// TwinCAT 3 PLC project Untitled1
// ProgramVersion: 3.1.4024.12
// libraries:
//   ActuatorMulti, * (Tesla)
//   Tc2_Standard, * (Beckhoff Automation GmbH)
//   Tc2_System, * (Beckhoff Automation GmbH)
//   Tc3_Module, * (Beckhoff Automation GmbH)
//   CycleHistory,1.2020.707.13,Tesla
//   E10Status,0.2020.423.6,Tesla
//   EM,0.2020.618.80,Tesla
//   Error,3.2020.227.2,Tesla
//   ExternalInterface,0.2020.610.18,Tesla
//   Input,7.2020.610.5,Tesla
//   LTU,5.2020.616.61,Tesla
//   NetworkDiagnostics,3.2020.617.20,Tesla
//   PalletStop,0.2020.609.18,Tesla
//   PermIntlk,3.2020.323.3,Tesla
//   PLC_Definition,5.2020.501.4,Tesla
//   Safety,3.2020.617.25,Tesla
//   Sequencer,2.2020.502.11,Tesla
//   Servo,3.2020.616.12,Tesla
//   TSM,3.2020.702.12,Tesla
//   VFD,2.2020.617.43,Tesla
//   ZoneManager,0.2020.429.17,Tesla
// project tree:
//   / PlcTask.TcTTO
//   Standard POUs/EquipmentModules/Conveyor/Enumerations/ E_ConveyorEMFixed.TcDUT, E_ConveyorEMTransition.TcDUT
//   Standard POUs/EquipmentModules/Conveyor/ FB_Conveyor_EM.TcPOU
//   Standard POUs/ MAIN.TcPOU
//   Standard POUs/TSM/ FB_SortingSystem_TSM.TcPOU
// real-time tasks:
//   TASK PlcTask: cycle T#10ms, priority 20, ADS port 350
// motion (NC):
//   TASK NC-Task 1 SAF: cycle T#2ms, priority 4, ADS port 501
//   TASK NC-Task 1 SVB: cycle T#10ms, priority 8, ADS port 511
//   AXIS Axis 1 (id 1)
//     Dynamic: Acceleration=6762, Deceleration=6762, Jerk=6762
//     Velo: RefSearch=135.24, RefSync=135.24, SlowManual=676.2, FastManual=4057.2, Fast=13524, Maximum=13524
//     OtherSettings: AllowMotionCmdToSlave=true
//     encoder EncType=19
//       EncPara: ScaleFactorNumerator=360, ScaleFactorDenominator=1048576, MaxCount=#xffffffff
//     drive DrvType=16
//       DrvPara: MaxCount=#xffffffff, DriveControlDWord=#x00020000
//         Analog: VeloReferenz=14876.4, VeloScale=32, TorqueSetpointScale=10, ScaleFactorActTorque=0.1
//         TimeComp: TaskDelayCycles=1
//     controller CtrType=1
//       CtrPara: PriorControlFactor=1
//         PosDiffControl: Range=25
//         Observer: BandWidth=20
//   AXIS Axis 2 (id 2)
//     OtherSettings: AllowMotionCmdToSlave=true
//     encoder EncType=8
//       EncPara: MaxCount=#xffffffff
//     drive DrvType=9
//       DrvPara: MaxCount=#xffffffff, DriveControlDWord=#x00030100
//         Analog: VeloScale=1.02400649589962, TorqueSetpointScale=10, ScaleFactorActTorque=0.1
//         TimeComp: TaskDelayCycles=1
//     controller CtrType=1
//       CtrPara: PriorControlFactor=1
//         Observer: BandWidth=20
//   AXIS Axis 3 (id 3)
//     Dynamic: Acceleration=53514.5668945313, Deceleration=53514.5668945313, Jerk=160543.700683594
//     Velo: RefSearch=356.763779296875, RefSync=356.763779296875, SlowManual=1783.81889648438, FastManual=10702.9133789062, Fast=35676.3779296875, Maximum=35676.3779296875
//     OtherSettings: AllowMotionCmdToSlave=true
//     encoder EncType=8
//       EncPara: ScaleFactorNumerator=360, ScaleFactorDenominator=1048576, MaxCount=#xffffffff
//     drive DrvType=9
//       DrvPara: MaxCount=#xffffffff, DriveControlDWord=#x00030100
//         Analog: VeloReferenz=39244.0157226563, VeloScale=1.02400649589962, TorqueSetpointScale=10, ScaleFactorActTorque=0.1
//         TimeComp: TaskDelayCycles=1
//     controller CtrType=1
//       CtrPara: PriorControlFactor=1
//         Observer: BandWidth=20
// I/O:
//   DEVICE Device 1 (EtherCAT), AmsNetId 5.79.65.80.2.1
//     Term 1 (EK1200) [EK1200-5000 EtherCAT Power supply (2A E-Bus)]
//       Term 2 (EL1819) [EL1819 16Ch. Dig. Input 24V, 10µs]
//       Term 3 (EL2809) [EL2809 16Ch. Dig. Output 24V, 0.5A]
//       Term 4 (EL3064) [EL3064 4Ch. Ana. Input 0-10V]
//       Term 5 (EL4004) [EL4004 4Ch. Ana. Output 0-10V, 12bit]
//       Term 6 (EL7201) [EL7201 1Ch. MDP742 Servo motor output stage (50V, 4A)]
//       Term 7 (EL9510) [EL9510 Power supply terminal 10V]
//       Term 8 (EL9011) [EL9011 End Terminal]
//   DEVICE Device 4 (EtherCAT), AmsNetId 5.79.65.80.5.1
//     Drive 9 (AX5203-0000-0203) [AX5203-0000-0203 EtherCAT Drive (SoE, 2 Ch.)]
//     Term 10 (EK1100) [EK1100 EtherCAT Coupler (2A E-Bus)]
//       Term 11 (EL6900) [EL6900, TwinSAFE PLC]
//       Term 12 (EL1904) [EL1904, 4 Ch. Safety Input 24V, TwinSAFE]
//         modules: Module 1 (FSOES)
//       Term 13 (EL1904) [EL1904, 4 Ch. Safety Input 24V, TwinSAFE]
//         modules: Module 1 (FSOES)
//       Term 14 (EL2904) [EL2904, 4 Ch. Safety Output 24V, 0.5A, TwinSAFE]
//         modules: Module 1 (FSOES), Module 2 (DO)
//       Term 7 (EL9011) [EL9011 End Terminal]
// variable links:
//   NC-Task 1 SAF/Axes/Axis 1 <-> Device 1 (EtherCAT)/Term 1 (EK1200)/Term 6 (EL7201)
//     Drive/Inputs/In/nDcOutputTime <-> InfoData/DcOutputShift
//     Drive/Inputs/In/nState1 <-> DRV Statusword/Statusword
//     Drive/Inputs/In/nState2 <-> DRV Statusword/Statusword @bit 8
//     Drive/Inputs/In/nState4 @bit 1 <-> WcState/InputToggle
//     Drive/Inputs/In/nState4 <-> WcState/WcState
//     Drive/Outputs/Out/nCtrl1 <-> DRV Controlword/Controlword
//     Drive/Outputs/Out/nCtrl2 <-> DRV Controlword/Controlword @bit 8
//     Drive/Outputs/Out/nDataOut2 <-> DRV Target velocity/Target velocity
//     Enc/Inputs/In/nDataIn1 <-> FB Position/Position
//     Enc/Inputs/In/nDcInputTime <-> InfoData/DcInputShift
//     Enc/Inputs/In/nState4 @bit 1 <-> WcState/InputToggle
//     Enc/Inputs/In/nState4 <-> WcState/WcState
//   NC-Task 1 SAF/Axes/Axis 2 <-> Device 4 (EtherCAT)/Drive 9 (AX5203-0000-0203)
//     Drive/Inputs/In/nDataIn1 <-> AT 1/Following distance
//     Drive/Inputs/In/nDcOutputTime <-> InfoData/DcOutputShift
//     Drive/Inputs/In/nState1 <-> AT 1/Drive status word @bit 8
//     Drive/Inputs/In/nState2 <-> AT 1/Drive status word
//     Drive/Inputs/In/nState4 @bit 1 <-> WcState/InputToggle
//     Drive/Inputs/In/nState4 <-> WcState/WcState
//     Drive/Outputs/Out/nCtrl1 <-> MDT 1/Master control word @bit 8
//     Drive/Outputs/Out/nDataOut1 <-> MDT 1/Position command value
//     Enc/Inputs/In/nDataIn1 <-> AT 1/Position feedback 1 value
//     Enc/Inputs/In/nDcInputTime <-> InfoData/DcInputShift
//     Enc/Inputs/In/nState4 @bit 1 <-> WcState/InputToggle
//     Enc/Inputs/In/nState4 <-> WcState/WcState
//   NC-Task 1 SAF/Axes/Axis 3 <-> Device 4 (EtherCAT)/Drive 9 (AX5203-0000-0203)
//     Drive/Inputs/In/nDataIn1 <-> AT 2/Following distance
//     Drive/Inputs/In/nDcOutputTime <-> InfoData/DcOutputShift
//     Drive/Inputs/In/nState1 <-> AT 2/Drive status word @bit 8
//     Drive/Inputs/In/nState2 <-> AT 2/Drive status word
//     Drive/Inputs/In/nState4 @bit 1 <-> WcState/InputToggle
//     Drive/Inputs/In/nState4 <-> WcState/WcState
//     Drive/Outputs/Out/nCtrl1 <-> MDT 2/Master control word @bit 8
//     Drive/Outputs/Out/nDataOut1 <-> MDT 2/Position command value
//     Enc/Inputs/In/nDataIn1 <-> AT 2/Position feedback 1 value
//     Enc/Inputs/In/nDcInputTime <-> InfoData/DcInputShift
//     Enc/Inputs/In/nState4 @bit 1 <-> WcState/InputToggle
//     Enc/Inputs/In/nState4 <-> WcState/WcState
//   Untitled1/Untitled1 Instance <-> NC-Task 1 SAF/Axes/Axis 1
//     PlcTask Inputs/MAIN.fbSortingSystemTSM.fbConveyorEM.fbConveyor.Axis.NcToPlc <-> Outputs/ToPlc
//     PlcTask Outputs/MAIN.fbSortingSystemTSM.fbConveyorEM.fbConveyor.Axis.PlcToNc <-> Inputs/FromPlc

CONFIGURATION Untitled1
    RESOURCE PLC ON TwinCAT3
        TASK PlcTask(INTERVAL := T#10ms, PRIORITY := 20);
        PROGRAM MAIN WITH PlcTask : MAIN;
    END_RESOURCE
END_CONFIGURATION

// ---- Standard POUs/EquipmentModules/Conveyor/Enumerations/E_ConveyorEMFixed.TcDUT
{attribute 'qualified_only'}
{attribute 'strict'}
TYPE E_ConveyorEMFixed :
(
	Stopped		:= 1,
	Running		:= 2,
	LastFixed	:= 3
);
END_TYPE

// ---- Standard POUs/EquipmentModules/Conveyor/Enumerations/E_ConveyorEMTransition.TcDUT
{attribute 'qualified_only'}
{attribute 'strict'}
TYPE E_ConveyorEMTransition :
(
	Starting		:= 1,
	Stopping		:= 2,
	Recovery		:= 3,
	LastTransition	:= 4
);
END_TYPE

// ---- Standard POUs/MAIN.TcPOU
PROGRAM MAIN
VAR
	fbSortingSystemTSM			: FB_SortingSystem_TSM;
END_VAR

// TSMs
	fbSortingSystemTSM();

END_PROGRAM

// ---- Standard POUs/TSM/FB_SortingSystem_TSM.TcPOU
FUNCTION_BLOCK FB_SortingSystem_TSM EXTENDS FB_TSM
VAR
	fbConveyorEM			: FB_Conveyor_EM;

	ButtonFaultReset    AT %I* : BOOL;
    ButtonStartProceed  AT %I* : BOOL;
    ButtonAbort         AT %I* : BOOL;
	ButtonRun			AT %I* : BOOL;
END_VAR

SUPER^();

// System Interlocks
    // The system interlock inherits the system interlock from the TSM's EMs OR from the safety zone. More interlocks can be added that are not part of the EM or safety zone interlocks.  
    SUPER^.P_SystemInterlock.M_Set(Index := 0, Description := 'Always TRUE' , Condition := TRUE);   // network devices OK

// Button Requests
    IF ButtonFaultReset THEN
        ButtonFaultReset := FALSE;
        SUPER^.M_Retry();
    ELSIF ButtonStartProceed THEN
        ButtonStartProceed := FALSE;
        SUPER^.M_Proceed();
    ELSIF ButtonAbort THEN
        ButtonAbort := FALSE;
        SUPER^.M_Abort();
    END_IF

// State Permissives
// Start
    SUPER^.P_StartPermissive.M_Set(index := 0, Description := 'FlipGantryEM in Fixed State', Condition := fbConveyorEM.P_Status.FixedStateIndex <> 0);
// Home
    SUPER^.P_HomePermissive.M_Set(index := 0, Description := 'Always TRUE', Condition := TRUE);
// Proceed
    SUPER^.P_ProceedPermissive.M_Set(index := 0, Description := 'Always TRUE', Condition := TRUE);

// Retry EMs on TSM Retry
    IF SUPER^.P_Status.Retry THEN
        fbConveyorEM.M_Retry();
	END_IF

// Equipment Modules
	M_ConveyorEM();

METHOD PROTECTED _M_Aborting
// Abort child Equipment Modules
    fbConveyorEM.M_Abort();

// Aborting Complete Permissives - Method will be cyclically executed until all permissives are met
    SUPER^.P_AbortCompletePermissive.M_Set(Index := 0,
										   Description := 'Conveyor Aborted',
										   Condition := fbConveyorEM.P_Status.StateStatus <> E_DeviceStatus.Active OR
														fbConveyorEM.P_Status.StateStatus <> E_DeviceStatus.Aborting);
END_METHOD

METHOD PROTECTED _M_Homing
//=========================================================================================
//    local constants
//=========================================================================================
VAR CONSTANT
    START                                                       : UDINT := 10;       // 10

    COMPLETE                                                    : UDINT := 1000;     // 1000
END_VAR
//=========================================================================================
//    local variables
//=========================================================================================
VAR_INST
    
END_VAR
// Set first step to 10
SUPER^.P_Configuration.HomingFirstStep := 10;

CASE SUPER^.P_HomingSequencer.P_Status.CurrentStep OF
	START:
        // Branch 0: At fixed state, skip PalletPositioner recovery and Finish
		SUPER^.P_HomingSequencer.M_SetBranchConfig(BranchIndex := 0, Description := 'No Recovery Needed', NextStep := COMPLETE, CheckWhileFaulted := TRUE);
		SUPER^.P_HomingSequencer.M_SetBranchPermissive(BranchIndex := 0,
                                                        PermissiveIndex := 0,
                                                        Description := 'At Fixed State',
                                                        Condition := fbConveyorEM.P_Status.FixedStateIndex <> 0);
	COMPLETE:
		_M_SeqComplete();
END_CASE
END_METHOD

METHOD PROTECTED _M_Pausing
VAR CONSTANT
    COMMAND_PAUSE : UDINT := 10;
	FINISH        : UDINT := 999;
END_VAR
// Set first step to 10
SUPER^.P_Configuration.PausingFirstStep := 10;

// Pausing Sequence
CASE SUPER^.P_PausingSequencer.P_Status.CurrentStep OF	
	COMMAND_PAUSE:
		CASE SUPER^.P_PausingSequencer.P_StepStatus.StepState OF
			E_StepState.ActiveEntry:
                // Set step configurations here
                SUPER^.P_PausingSequencer.P_StepConfig.Name := 'Pause EMs';
				SUPER^.P_PausingSequencer.P_StepConfig.Timeout := T#15S; // Optional step timeout. Set to zero to ignore
                // Issue EM commands here
				    fbConveyorEM.M_Pause();
			E_StepState.ActiveDuring:
                // Check for errors on EMs commanded on this step here
				SUPER^.P_PausingSequencer.M_CheckFaultCondition(Error := fbConveyorEM.P_Error);
            E_StepState.ActiveExit:
                //
            E_StepState.FaultedEntry:
                //
            E_StepState.FaultedDuring:
                //
            E_StepState.FaultedExit:
                //
        END_CASE
        // Branch 0: EMs Paused Successfully
		SUPER^.P_PausingSequencer.M_SetBranchConfig(BranchIndex := 0, Description := 'EMs Paused Successfully', NextStep := FINISH, CheckWhileFaulted := TRUE);
		SUPER^.P_PausingSequencer.M_SetBranchPermissive(BranchIndex := 0,
                                                           PermissiveIndex := 0,
                                                           Description := 'fbConveyorEM Paused OR Complete',
                                                           Condition := fbConveyorEM.P_Status.StateStatus = E_DeviceStatus.Paused OR
                                                                        fbConveyorEM.P_Status.StateStatus = E_DeviceStatus.Complete);                                                 
        
	FINISH:
        // Sequence must end with the following method call
		_M_SeqComplete(); 
END_CASE
END_METHOD

METHOD PROTECTED _M_Proceeding
VAR CONSTANT
    COMMAND_PROCEED : UDINT := 10;
	FINISH          : UDINT := 999;
END_VAR
// Set first step to 10
SUPER^.P_Configuration.ProceedingFirstStep := 10;

// Proceeding Sequence
CASE SUPER^.P_ProceedingSequencer.P_Status.CurrentStep OF	
	COMMAND_PROCEED:
		CASE SUPER^.P_ProceedingSequencer.P_StepStatus.StepState OF
			E_StepState.ActiveEntry:
                // Set step configurations here
                SUPER^.P_ProceedingSequencer.P_StepConfig.Name := 'Proceed EMs';
				SUPER^.P_ProceedingSequencer.P_StepConfig.Timeout := T#15S; // Optional step timeout. Set to zero to ignore
                // Issue EM commands here
				    fbConveyorEM.M_Proceed();
			E_StepState.ActiveDuring:
                // Check for errors on EMs commanded on this step here
				SUPER^.P_ProceedingSequencer.M_CheckFaultCondition(Error := fbConveyorEM.P_Error);
            E_StepState.ActiveExit:
                //
            E_StepState.FaultedEntry:
                //
            E_StepState.FaultedDuring:
                //
            E_StepState.FaultedExit:
                //
        END_CASE
        // Branch 0: EMs Proceeded Successfully
		SUPER^.P_ProceedingSequencer.M_SetBranchConfig(BranchIndex := 0, Description := 'EMs Proceeded Successfully', NextStep := FINISH, CheckWhileFaulted := TRUE);
		SUPER^.P_ProceedingSequencer.M_SetBranchPermissive(BranchIndex := 0,
                                                           PermissiveIndex := 0,
                                                           Description := 'fbConveyorEM Active OR Complete',
                                                           Condition := fbConveyorEM.P_Status.StateStatus = E_DeviceStatus.Active OR
                                                                        fbConveyorEM.P_Status.StateStatus = E_DeviceStatus.Complete);                                                    
        
	FINISH:
        // Sequence must end with the following method call
		_M_SeqComplete(); 
END_CASE
END_METHOD

METHOD PROTECTED _M_Running
VAR CONSTANT
    START_BRANCH	: UDINT := 10;
    START			: UDINT := 20;
	RUNNING			: UDINT := 30;
	STOP			: UDINT := 40;
	FINISH			: UDINT := 999;
END_VAR
// Set first step to 10
SUPER^.P_Configuration.RunningFirstStep := 10;

CASE SUPER^.P_RunningSequencer.P_Status.CurrentStep OF
	START_BRANCH:
        // Branch 0:
		SUPER^.P_RunningSequencer.M_SetBranchConfig(BranchIndex := 0, Description := 'Conveyor START', NextStep := START, CheckWhileFaulted := TRUE);
		SUPER^.P_RunningSequencer.M_SetBranchPermissive(BranchIndex := 0,
                                                        PermissiveIndex := 0,
                                                        Description := 'EM at Stopped',
                                                        Condition := fbConveyorEM.P_Status.FixedStateIndex = E_ConveyorEMFixed.Stopped);
		SUPER^.P_RunningSequencer.M_SetBranchPermissive(BranchIndex := 0,
                                                        PermissiveIndex := 1,
                                                        Description := 'ButtonRun is TRUE',
                                                        Condition := ButtonRun);

        // Branch 1:
		SUPER^.P_RunningSequencer.M_SetBranchConfig(BranchIndex := 1, Description := 'Conveyor Running', NextStep := RUNNING, CheckWhileFaulted := TRUE);
		SUPER^.P_RunningSequencer.M_SetBranchPermissive(BranchIndex := 1,
                                                        PermissiveIndex := 0,
                                                        Description := 'EM at Running',
                                                        Condition := fbConveyorEM.P_Status.FixedStateIndex = E_ConveyorEMFixed.Running);
    START:
        CASE SUPER^.P_RunningSequencer.P_StepStatus.StepState OF
			E_StepState.ActiveEntry:
                // Set step configurations here
                SUPER^.P_RunningSequencer.P_StepConfig.Name := 'Command EM to Run Conveyor';
				SUPER^.P_RunningSequencer.P_StepConfig.Timeout := T#5S; // Optional step timeout. Set to zero to ignore
                SUPER^.P_RunningSequencer.P_StepConfig.IgnoreHold := FALSE; // This step is pausable.
                SUPER^.P_RunningSequencer.P_StepConfig.NextStepAfterRetry := 0; // Optional.  Set to zero to ignore
                // Issue EM commands here
                    fbConveyorEM.M_TransitionNumberRequest(E_ConveyorEMTransition.Starting);
			E_StepState.ActiveDuring:
                // Check for errors on EMs commanded on this step here
                SUPER^.P_RunningSequencer.M_CheckFaultCondition(Error := fbConveyorEM.P_Error);
            E_StepState.ActiveExit:
                //
            E_StepState.FaultedEntry:
                //
            E_StepState.FaultedDuring:
                //
            E_StepState.FaultedExit:
                //
        END_CASE
		// Branch 0: EMs Proceeded Successfully
		SUPER^.P_RunningSequencer.M_SetBranchConfig(BranchIndex := 0, Description := 'ConveyorEM Transition Finished', NextStep := RUNNING, CheckWhileFaulted := TRUE);
		SUPER^.P_RunningSequencer.M_SetBranchPermissive(BranchIndex := 0,
                                                        PermissiveIndex := 0,
                                                        Description := 'EM at Running',
                                                        Condition := fbConveyorEM.P_Status.FixedStateIndex = E_ConveyorEMFixed.Running);
    RUNNING:
        CASE SUPER^.P_RunningSequencer.P_StepStatus.StepState OF
			E_StepState.ActiveEntry:
                // Set step configurations here
                SUPER^.P_RunningSequencer.P_StepConfig.Name := 'Command EM to Run Conveyor';
				SUPER^.P_RunningSequencer.P_StepConfig.Timeout := T#0S; // Optional step timeout. Set to zero to ignore
                SUPER^.P_RunningSequencer.P_StepConfig.IgnoreHold := FALSE; // This step is pausable.
                SUPER^.P_RunningSequencer.P_StepConfig.NextStepAfterRetry := 0; // Optional.  Set to zero to ignore
                // Issue EM commands here
			E_StepState.ActiveDuring:
                // Check for errors on EMs commanded on this step here
                SUPER^.P_RunningSequencer.M_CheckFaultCondition(Error := fbConveyorEM.P_Error);
            E_StepState.ActiveExit:
                //
            E_StepState.FaultedEntry:
                //
            E_StepState.FaultedDuring:
                //
            E_StepState.FaultedExit:
                //
        END_CASE
		// Branch 0: EMs Proceeded Successfully
		SUPER^.P_RunningSequencer.M_SetBranchConfig(BranchIndex := 0, Description := 'TSM Received Complete Signal', NextStep := STOP, CheckWhileFaulted := TRUE);
		SUPER^.P_RunningSequencer.M_SetBranchPermissive(BranchIndex := 0,
                                                        PermissiveIndex := 0,
                                                        Description := 'ButtonRun is FALSE',
                                                        Condition := NOT ButtonRun);
    STOP:
        CASE SUPER^.P_RunningSequencer.P_StepStatus.StepState OF
			E_StepState.ActiveEntry:
                // Set step configurations here
                SUPER^.P_RunningSequencer.P_StepConfig.Name := 'Command EM to Run Conveyor';
				SUPER^.P_RunningSequencer.P_StepConfig.Timeout := T#5S; // Optional step timeout. Set to zero to ignore
                SUPER^.P_RunningSequencer.P_StepConfig.IgnoreHold := FALSE; // This step is pausable.
                SUPER^.P_RunningSequencer.P_StepConfig.NextStepAfterRetry := 0; // Optional.  Set to zero to ignore
                // Issue EM commands here
                    fbConveyorEM.M_TransitionNumberRequest(E_ConveyorEMTransition.Stopping);
			E_StepState.ActiveDuring:
                // Check for errors on EMs commanded on this step here
                SUPER^.P_RunningSequencer.M_CheckFaultCondition(Error := fbConveyorEM.P_Error);
            E_StepState.ActiveExit:
                //
            E_StepState.FaultedEntry:
                //
            E_StepState.FaultedDuring:
                //
            E_StepState.FaultedExit:
                //
        END_CASE
		// Branch 0: EMs Proceeded Successfully
		SUPER^.P_RunningSequencer.M_SetBranchConfig(BranchIndex := 0, Description := 'ConveyorEM Transition Finished', NextStep := FINISH, CheckWhileFaulted := TRUE);
		SUPER^.P_RunningSequencer.M_SetBranchPermissive(BranchIndex := 0,
                                                        PermissiveIndex := 0,
                                                        Description := 'EM at Stopped',
                                                        Condition := fbConveyorEM.P_Status.FixedStateIndex = E_ConveyorEMFixed.Stopped);
	FINISH:
        // Sequence must end with the following method call
		_M_SeqComplete(); 
END_CASE
END_METHOD

METHOD M_ConveyorEM
// Set System Interlocks
// Index 0 is set in EM FB

// Call EM
    fbConveyorEM();
END_METHOD

END_FUNCTION_BLOCK

// ---- Standard POUs/EquipmentModules/Conveyor/FB_Conveyor_EM.TcPOU
FUNCTION_BLOCK FB_Conveyor_EM EXTENDS FB_EquipmentModule
VAR
	// Devices
	fbConveyor				: FB_Servo;
	ConveyorMoves			: ARRAY[1..1] OF ST_ServoMove;
	ConveyorMoveTolerance	: LREAL := 0.1;
	
	ConveyorTransitionStates	: ARRAY[E_ConveyorEMFixed.Stopped..E_ConveyorEMFixed.LastFixed] OF ST_EmTransitionState;
	ConveyorFixedStates			: ARRAY[E_ConveyorEMTransition.Starting..E_ConveyorEMTransition.LastTransition] OF ST_EmFixedState;
	UnknownTransitions			: ARRAY[1..Param_EquipmentModule.MAX_TRANSITIONS] OF ST_TransitionDefinition;

	//First Scan Bit for configurations
	FirstScan					: BOOL := TRUE;
END_VAR

// Configuration
IF FirstScan THEN
    SUPER^.P_Configuration.Definition.description  := 'Conveyor to move boxes';
    SUPER^.P_Configuration.Definition.deviceType   := 'Equipment Module';
    SUPER^.P_Configuration.Definition.displayName  := 'ConveyorEM';
    SUPER^.P_Configuration.Definition.parentName   := 'IDK';
    SUPER^.P_Configuration.Definition.categoryName := 'EM';
END_IF

// Call Body of Super Class
    SUPER^(TransitionStates := ConveyorTransitionStates, FixedStates := ConveyorFixedStates);

// Configure Unknown Transitions
    UnknownTransitions[1].Name    := ConveyorTransitionStates[E_ConveyorEMTransition.Stopping].Name;
    UnknownTransitions[1].Command := ConveyorTransitionStates[E_ConveyorEMTransition.Stopping].Command;
    UnknownTransitions[1].Target  := ConveyorTransitionStates[E_ConveyorEMTransition.Stopping].Target;
	
	SUPER^.P_Configuration.UnknownTransitions := UnknownTransitions;

// System Interlocks
    // The system interlock inherits the interlock from the safety zone OR from its child devices (ex: Actuator)
	SUPER^.P_SystemInterlock.M_Set(Index := 0, Description := 'Always TRUE', Condition := TRUE);  

// Control Devices
	_M_Conveyor();

// Fixed States
	_M_Running();
	_M_Stopped();

// Transition States
	_M_Starting();
	_M_Stopping();

// Unknown Transitions
	

FirstScan := FALSE;

METHOD PROTECTED _M_Aborting
// Aborting Complete Permissives - Method will be cyclically executed until all permissives are met
    //Typically, stop commands will be executed to some or all control devices and a permissive will set for each device checking it is stopped or idle
fbConveyor.M_Stop(0, 0);

SUPER^.fbAbortingCompletePermissive.M_Set(Index := 0, Description := 'Conveyor is Stopped', Condition := fbConveyor.P_Status.idle);
END_METHOD

METHOD _M_Conveyor
//All devices are defined & initialized in the Main FB
//Use 1 Method per device to combine all device configurations and device FB call

//Configuration
IF FirstScan THEN
    //General Configuration
	fbConveyor.P_Configuration.Definition.displayName  := 'Z Servo';
	fbConveyor.P_Configuration.Definition.description  := 'Flipper Gantry Servo';
	fbConveyor.P_Configuration.Definition.parentName   := 'FlipGantryEM';
	fbConveyor.P_Configuration.Definition.categoryName := 'Device';
	fbConveyor.P_Configuration.Definition.deviceType   := 'Servo';

    fbConveyor.P_Configuration.SafetyStopDeceleration := 0; // Using 0 forces it to use the deceleration of the previous/active command
    fbConveyor.P_Configuration.SafetyStopJerk := 0; // Using 0 forces it to use the jerk of the previous/active command
END_IF

// Setup Servo Moves Array
ConveyorMoves[1].Name := 'Run';
ConveyorMoves[1].Acceleration := 500;
ConveyorMoves[1].Deceleration := 500;
ConveyorMoves[1].Direction := 1;
ConveyorMoves[1].Jerk := 5000;
ConveyorMoves[1].MoveType := E_ServoMoveType.Velocity;
ConveyorMoves[1].Velocity := 500;
ConveyorMoves[1].Permissive.M_Set(Index := 0, Description := '', Condition := TRUE);

fbConveyor(Moves := ConveyorMoves);
END_METHOD

METHOD PROTECTED _M_Pausing
VAR CONSTANT
    PAUSE		: UDINT := 10;
    FINISH		: UDINT := 999;
END_VAR
//Method can be used to send commands to devices either directly or using a built in sequencer (fbPausingSequencer)
SUPER^.fbPausingSequencer.P_Config.FirstStep := PAUSE;

// Pausing Sequence
CASE SUPER^.fbPausingSequencer.P_Status.CurrentStep OF
	PAUSE:
		CASE SUPER^.fbPausingSequencer.P_StepStatus.StepState OF
			E_StepState.ActiveEntry:
                // Set step configurations here
                SUPER^.fbPausingSequencer.P_StepConfig.Name := 'Pause Conveyor';
				SUPER^.fbPausingSequencer.P_StepConfig.Timeout := T#15S; // Optional step timeout. Set to zero to ignore
                SUPER^.fbPausingSequencer.P_StepConfig.IgnoreHold := FALSE; // This step is pausable.
                SUPER^.fbPausingSequencer.P_StepConfig.NextStepAfterRetry := 0; // Optional.  Set to zero to ignore
                // Issue device commands here
					fbConveyor.M_Halt(0, 0);
			E_StepState.ActiveDuring:
                // Check for errors on devices commanded on this step here
				SUPER^.fbPausingSequencer.M_CheckFaultCondition(Error := fbConveyor.P_Error);
            E_StepState.ActiveExit:
                //
            E_StepState.FaultedEntry:
                //
            E_StepState.FaultedDuring:
                //
            E_StepState.FaultedExit:
                //
        END_CASE
        // Branch 0: Conveyor VFD paused successfully
		SUPER^.fbPausingSequencer.M_SetBranchConfig(BranchIndex := 0, Description := 'Conveyor is Stopped', NextStep := FINISH, CheckWhileFaulted := TRUE);
		SUPER^.fbPausingSequencer.M_SetBranchPermissive(BranchIndex := 0, PermissiveIndex := 0, Description := 'Conveyor is Stopped', Condition := fbConveyor.P_Status.Idle);
	FINISH:
        //Method will be cyclically executed until the following method is executed
		M_PausingComplete();
END_CASE
END_METHOD

METHOD PROTECTED _M_Proceeding
M_ProceedingComplete();
END_METHOD

METHOD _M_Recovery
VAR_INST
	State	        : REFERENCE TO ST_EmTransitionState;
END_VAR
VAR CONSTANT
	START	: UDINT := 10;
	RESET	: UDINT := 20;
	FINISH	: UDINT := 999;
END_VAR
// Set Reference
State REF= THIS^.ConveyorTransitionStates[E_ConveyorEMTransition.Recovery];

// Name this Transition State
	State.Name := 'Recovery';
	State.Command := 'Recovery';
	State.Target := THIS^.ConveyorFixedStates[E_ConveyorEMFixed.Stopped].Name;

// Permissives that must be met in order to call this Transition State
	State.fbPermissive.M_Set(Index := 0, Description := 'ALWAYS TRUE', Condition := TRUE);
	
// Set first step to 10
	State.fbSequencer.P_Config.FirstStep := 10;

// Sequence
    CASE State.fbSequencer.P_Status.CurrentStep OF
		START:
			CASE state.fbSequencer.P_StepStatus.StepState OF
				E_StepState.ActiveEntry:
                    // Set step configurations here
                    State.fbSequencer.P_StepConfig.Name := 'Conveyor Halt';
                    State.fbSequencer.P_StepConfig.Timeout := T#10S; // Optional step timeout. Set to zero to ignore
                    State.fbSequencer.P_StepConfig.IgnoreHold := FALSE; // This step is pausable.
                    State.fbSequencer.P_StepConfig.NextStepAfterRetry := RESET; // Optional.  Set to zero to ignore
                    // Issue device commands here
					fbConveyor.M_Halt(0, 0);
                E_StepState.ActiveDuring:
					// Check for errors on devices commanded on this step here
                    State.fbSequencer.M_CheckFaultCondition(Error := fbConveyor.P_Error);
                E_StepState.ActiveExit:
                    //
                E_StepState.FaultedEntry:
                    //
                E_StepState.FaultedDuring:
                    //
                E_StepState.FaultedExit:
                    //
			END_CASE
            // Branch 0: Conveyor Halted Successfully
                State.fbSequencer.M_SetBranchConfig(BranchIndex := 0, Description := 'Conveyor Halted', NextStep := FINISH, CheckWhileFaulted := FALSE);
                State.fbSequencer.M_SetBranchPermissive(BranchIndex := 0,
														PermissiveIndex := 0,
														Description := 'Conveyor Halted',
														Condition := NOT fbConveyor.P_Status.Busy AND fbConveyor.P_Status.Idle);
		RESET:
            CASE State.fbSequencer.P_StepStatus.StepState OF
                E_StepState.ActiveEntry:
                    // Set step configurations here
                    State.fbSequencer.P_StepConfig.Name := 'Conveyor Reset';
                    State.fbSequencer.P_StepConfig.Timeout := T#10S; // Optional step timeout. Set to zero to ignore
                    State.fbSequencer.P_StepConfig.IgnoreHold := FALSE; // This step is pausable.
                    State.fbSequencer.P_StepConfig.NextStepAfterRetry := 0; // Optional.  Set to zero to ignore
                    // Issue device commands here
                    fbConveyor.M_Reset();
                E_StepState.ActiveDuring:
					// Check for errors on devices commanded on this step here
					State.fbSequencer.M_CheckFaultCondition(Error := fbConveyor.P_Error);
                E_StepState.ActiveExit:
                    //
                E_StepState.FaultedEntry:
                    //
                E_StepState.FaultedDuring:
                    //
                E_StepState.FaultedExit:
                    //
            END_CASE
            // Branch 0: Conveyor Reset
                State.fbSequencer.M_SetBranchConfig(BranchIndex := 0, Description := 'Conveyor Reset', NextStep := START, CheckWhileFaulted := FALSE);
                State.fbSequencer.M_SetBranchPermissive(BranchIndex := 0,
														PermissiveIndex := 0,
														Description := 'Conveyor is not Resetting',
														Condition := NOT fbConveyor.P_Status.Resetting);
                State.fbSequencer.M_SetBranchPermissive(BranchIndex := 0,
														PermissiveIndex := 1,
														Description := 'Conveyor No Error',
														Condition := NOT fbConveyor.P_Error.Active);
		FINISH:
            // Each sequence must end with the following method call
            M_TransitionComplete();
	END_CASE
END_METHOD

METHOD _M_Running
VAR_INST
	State	: REFERENCE TO ST_EmFixedState;
END_VAR
// Set Reference
State REF= THIS^.ConveyorFixedStates[E_ConveyorEMFixed.Running];

// Name this Fixed State
    State.Name := 'Running';

// Identify which transitions can be called from this Fixed State, index starting at 1
    // Transition 1: Stopping
        State.Transitions[1].Name    := THIS^.ConveyorTransitionStates[E_ConveyorEMTransition.Stopping].Name;
        State.Transitions[1].Command := THIS^.ConveyorTransitionStates[E_ConveyorEMTransition.Stopping].Command;
        State.Transitions[1].Target  := THIS^.ConveyorTransitionStates[E_ConveyorEMTransition.Stopping].Target;

// Interlocks that must be met to be in this Fixed State
	State.fbInterlock.M_Set(Index := 0, Description := 'Axis velocity is constant', Condition := fbConveyor.P_Status.ConstantVelocity);
END_METHOD

METHOD _M_Starting
VAR_INST
	State	: REFERENCE TO ST_EmTransitionState;
END_VAR
VAR CONSTANT
	START	: UDINT := 10;
	FINISH	: UDINT := 999;
END_VAR
// Set Reference
State REF= THIS^.ConveyorTransitionStates[E_ConveyorEMTransition.Starting];

// Name this Transition State
	State.Name := 'Starting';
	State.Command := 'Starting';
	State.Target := THIS^.ConveyorFixedStates[E_ConveyorEMFixed.Running].Name;

// Permissives that must be met in order to call this Transition State
// These permissives are anything that isn't covered by user configured allowed transitions from Fixed and Unknown states
	State.fbPermissive.M_Set(Index := 0, Description := 'ALWAYS TRUE', Condition := TRUE);

// Set first step to 10
	State.fbSequencer.P_Config.FirstStep := 10;

// Sequence
    CASE State.fbSequencer.P_Status.CurrentStep OF
		START:
			CASE State.fbSequencer.P_StepStatus.StepState OF
				E_StepState.ActiveEntry:
                    // Set step configurations here
                    State.fbSequencer.P_StepConfig.Name := 'Rotate Conveyor Belt to Move Box';
                    State.fbSequencer.P_StepConfig.Timeout := T#0S; // Optional step timeout. Set to zero to ignore
                    State.fbSequencer.P_StepConfig.IgnoreHold := FALSE; // This step is pausable.
                    State.fbSequencer.P_StepConfig.NextStepAfterRetry := 0; // Optional.  Set to zero to ignore
                    // Issue device commands here
					fbConveyor.M_Move(1);
				E_StepState.ActiveDuring:
                    // Check for errors on devices commanded on this step here
                    State.fbSequencer.M_CheckFaultCondition(Error := fbConveyor.P_Error);
				E_StepState.ActiveExit:
					;
				E_StepState.FaultedEntry:
					;
				E_StepState.FaultedDuring:
					;
				E_StepState.FaultedExit:
					;
			END_CASE
			// Branch 0: Actuator Advanced Successfully
				State.fbSequencer.M_SetBranchConfig(BranchIndex := 0, Description := '', NextStep := FINISH, CheckWhileFaulted := TRUE);
				state.fbSequencer.M_SetBranchPermissive(BranchIndex := 0, PermissiveIndex := 0, Description := '', Condition := fbConveyor.P_Status.ConstantVelocity);
		FINISH:
            // Each sequence must end with the following method call
            M_TransitionComplete();
	END_CASE
END_METHOD

METHOD _M_Stopped
VAR_INST
	State	: REFERENCE TO ST_EmFixedState;
END_VAR
// Set Reference
State REF= THIS^.ConveyorFixedStates[E_ConveyorEMFixed.Stopped];

// Name this Fixed State
    State.Name := 'Stopped';

// Identify which transitions can be called from this Fixed State, index starting at 1
    // Transition 1: Starting
        State.Transitions[1].Name    := THIS^.ConveyorTransitionStates[E_ConveyorEMTransition.Starting].Name;
        State.Transitions[1].Command := THIS^.ConveyorTransitionStates[E_ConveyorEMTransition.Starting].Command;
        State.Transitions[1].Target  := THIS^.ConveyorTransitionStates[E_ConveyorEMTransition.Starting].Target;

// Interlocks that must be met to be in this Fixed State
	State.fbInterlock.M_Set(Index := 0, Description := 'Axis is not moving', Condition := NOT fbConveyor.P_Status.Moving);
END_METHOD

METHOD _M_Stopping
VAR_INST
	State	: REFERENCE TO ST_EmTransitionState;
END_VAR
VAR CONSTANT
	STOP	: UDINT := 10;
	FINISH	: UDINT := 999;
END_VAR
// Set Reference
State REF= THIS^.ConveyorTransitionStates[E_ConveyorEMTransition.Stopping];

// Name this Transition State
	State.Name := 'Stopping';
	State.Command := 'Stopping';
	State.Target := THIS^.ConveyorFixedStates[E_ConveyorEMFixed.Stopped].Name;

// Permissives that must be met in order to call this Transition State
// These permissives are anything that isn't covered by user configured allowed transitions from Fixed and Unknown states
	State.fbPermissive.M_Set(Index := 0, Description := 'ALWAYS TRUE', Condition := TRUE);

// Set first step to 10
	State.fbSequencer.P_Config.FirstStep := 10;

// Sequence
    CASE State.fbSequencer.P_Status.CurrentStep OF
		STOP:
			CASE State.fbSequencer.P_StepStatus.StepState OF
				E_StepState.ActiveEntry:
                    // Set step configurations here
                    State.fbSequencer.P_StepConfig.Name := 'Stop Conveyor Belt';
                    State.fbSequencer.P_StepConfig.Timeout := T#0S; // Optional step timeout. Set to zero to ignore
                    State.fbSequencer.P_StepConfig.IgnoreHold := FALSE; // This step is pausable.
                    State.fbSequencer.P_StepConfig.NextStepAfterRetry := 0; // Optional.  Set to zero to ignore
                    // Issue device commands here
					fbConveyor.M_Halt(0, 0);
				E_StepState.ActiveDuring:
                    // Check for errors on devices commanded on this step here
                    State.fbSequencer.M_CheckFaultCondition(Error := fbConveyor.P_Error);
				E_StepState.ActiveExit:
					;
				E_StepState.FaultedEntry:
					;
				E_StepState.FaultedDuring:
					;
				E_StepState.FaultedExit:
					;
			END_CASE
			// Branch 0: Actuator Advanced Successfully
				State.fbSequencer.M_SetBranchConfig(BranchIndex := 0, Description := '', NextStep := FINISH, CheckWhileFaulted := TRUE);
				state.fbSequencer.M_SetBranchPermissive(BranchIndex := 0, PermissiveIndex := 0, Description := '', Condition := fbConveyor.P_Status.ConstantVelocity);
		FINISH:
            // Each sequence must end with the following method call
            M_TransitionComplete();
	END_CASE
END_METHOD

END_FUNCTION_BLOCK
